FUNCTION_BLOCK CLIENT_2_1
  (* Standard: 61499-2; Description: Copyright (c) 2017 fortiss GmbH This program and the accompanying materials are made available under the terms of the Eclipse Public License 2.0 which is available at https://www.eclipse.org/legal/epl-2.0/ SPDX-License-Identifier: EPL-2.0 *)
  (* Version 1.0, 2017-10-25, Alois Zoitl, fortiss GmbH, initial API and implementation and/or initial documentation *)
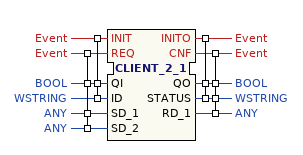
  EVENT_INPUT
    INIT WITH QI, ID;
    REQ WITH QI, SD_1, SD_2;
  END_EVENT
  EVENT_OUTPUT
    INITO WITH QO, STATUS;
    CNF WITH QO, STATUS, RD_1;
  END_EVENT
  VAR_INPUT
    QI : BOOL;
    ID : WSTRING;
    SD_1 : ANY;
    SD_2 : ANY;
  END_VAR
  VAR_OUTPUT
    QO : BOOL;
    STATUS : WSTRING;
    RD_1 : ANY;
  END_VAR
END_FUNCTION_BLOCK
